// TwinCAT 3 PLC project Panels
// ProgramVersion: 3.1.4026.20
// libraries:
//   Core, * (Beckhoff Automation LLC)
//   CoreComponents, * (Beckhoff Automation LLC)
//   CoreMotionNc2, * (Beckhoff Automation LLC)
//   Mechatronics Core, * (Beckhoff Automation LLC)
//   Tc2_Standard, * (Beckhoff Automation GmbH)
//   Tc2_System, * (Beckhoff Automation GmbH)
//   Xts Core, * (Beckhoff Automation LLC)
// project tree:
//   DUTs/ ST_Chiller_HMI.TcDUT, ST_Compressor_HMI.TcDUT, ST_Conveyor_HMI.TcDUT, ST_CuringOven_HMI.TcDUT, ST_Dispenser_HMI.TcDUT, ST_EStop_HMI.TcDUT, ST_HeaterCooler_HMI.TcDUT, ST_IndexingTable_HMI.TcDUT, ST_InterlockChain_HMI.TcDUT, ST_LightCurtain_HMI.TcDUT, ST_MixingStation_HMI.TcDUT, ST_NetworkSwitch_HMI.TcDUT, ST_LocalLog.TcDUT, ST_PidController_HMI.TcDUT, ST_PeekerEntry.TcDUT, ST_PickAndPlaceUnit_HMI.TcDUT, ST_Pump_HMI.TcDUT, ST_Robot_HMI.TcDUT, ST_SafetyDoor_HMI.TcDUT, ST_UPS_HMI.TcDUT, ST_Valve_HMI.TcDUT, ST_VFD_HMI.TcDUT, ST_Vision_HMI.TcDUT, ST_XtsSystem_HMI.TcDUT, ST_XtsMover_HMI.TcDUT, ST_XtsStation_HMI.TcDUT, ST_XtsPositionTrigger_HMI.TcDUT, ST_XtsZone_HMI.TcDUT
//   / PlcTask.TcTTO
//   POUs/ MAIN.TcPOU
// real-time tasks:
//   TASK PlcTask: cycle T#10ms, priority 20, ADS port 350

CONFIGURATION Panels
    RESOURCE PLC ON TwinCAT3
        TASK PlcTask(INTERVAL := T#10ms, PRIORITY := 20);
        PROGRAM MAIN WITH PlcTask : MAIN;
    END_RESOURCE
END_CONFIGURATION

// ---- DUTs/ST_Chiller_HMI.TcDUT
TYPE ST_Chiller_HMI EXTENDS ST_HmiFunction :
STRUCT

    // Display Parameters - Panel Data Points
    Temperature         : LREAL;        // Current outlet temperature in °C
    FlowRate            : LREAL;        // Current flow rate in L/min

    // Display Parameters - Popup Data Points
    TemperatureSetpoint : LREAL;        // Temperature setpoint in °C
    AlarmStatus         : BOOL;         // Alarm condition present
    InletTemperature    : LREAL;        // Inlet temperature in °C

    // Status Indicators
    Running             : BOOL;         // Chiller is running
    Enabled             : BOOL;         // Chiller is enabled
    HasFault            : BOOL;         // Fault condition present
    AtSetpoint          : BOOL;         // Target setpoint reached
    LowFlowAlarm        : BOOL;         // Low flow alarm active

    // Fault Information
    ErrorId             : DINT;         // Active error code

    // Control Setpoints
    TargetTemperature   : LREAL;        // Target temperature setpoint in °C
    TargetFlowRate      : LREAL;        // Target flow rate in L/min
    MinTemperature      : LREAL;        // Minimum temperature limit in °C
    MaxTemperature      : LREAL;        // Maximum temperature limit in °C

    // Command Buttons (rising edge triggered)
    Start               : Button;       // Start chiller command
    Stop                : Button;       // Stop chiller command
    Reset               : Button;       // Reset fault command

    // Statistics
    TotalRuntime        : LREAL;        // Total runtime in hours
    TotalStarts         : UDINT;        // Total number of starts
    AvgTemperature      : LREAL;        // Average temperature in °C
    AvgFlowRate         : LREAL;        // Average flow rate in L/min
    TotalCoolingEnergy  : LREAL;        // Total cooling energy in kWh
    AlarmCount          : UDINT;        // Total number of alarms

END_STRUCT
END_TYPE

// ---- DUTs/ST_Compressor_HMI.TcDUT
TYPE ST_Compressor_HMI EXTENDS ST_HmiFunction :
STRUCT

    // Display Parameters - Panel Data Points
    Pressure            : LREAL;        // Current pressure in bar
    Runtime             : LREAL;        // Current runtime in hours

    // Display Parameters - Popup Data Points
    MaintenanceInterval : LREAL;        // Next maintenance in hours
    Temperature         : LREAL;        // Current temperature in °C

    // Status Indicators
    Running             : BOOL;         // Compressor is running
    Enabled             : BOOL;         // Compressor is enabled
    HasFault            : BOOL;         // Fault condition present
    AtPressure          : BOOL;         // Target pressure reached
    OverTemperature     : BOOL;         // Temperature limit exceeded

    // Fault Information
    ErrorId             : DINT;         // Active error code

    // Control Setpoints
    TargetPressure      : LREAL;        // Target pressure setpoint in bar
    MaxPressure         : LREAL;        // Maximum pressure limit in bar
    MinPressure         : LREAL;        // Minimum pressure limit in bar
    MaxTemperature      : LREAL;        // Maximum temperature limit in °C

    // Command Buttons (rising edge triggered)
    Start               : Button;       // Start compressor command
    Stop                : Button;       // Stop compressor command
    Reset               : Button;       // Reset fault command

    // Statistics
    TotalStarts         : UDINT;        // Total number of starts
    TotalRuntime        : LREAL;        // Total runtime in hours
    AvgPressure         : LREAL;        // Average pressure in bar
    AvgTemperature      : LREAL;        // Average temperature in °C
    LastMaintenanceDate : STRING;       // Last maintenance date/time
    HoursToMaintenance  : LREAL;        // Hours remaining until maintenance

END_STRUCT
END_TYPE

// ---- DUTs/ST_Conveyor_HMI.TcDUT
TYPE ST_Conveyor_HMI EXTENDS ST_HmiFunction :
STRUCT

	// Status Information
    Running                 : BOOL;           // Conveyor is currently running
    Enabled                 : BOOL;           // Conveyor is enabled
    AutoMode                : BOOL;           // Operating in automatic mode
    JamDetected             : BOOL;           // Jam condition detected
    ReverseDirection        : BOOL;           // Currently running in reverse direction

    // Error Information
    HasError                : BOOL;           // Error condition present
    ErrorCode               : UDINT;          // Specific error code

    // Speed and Motor Information
    ActualSpeed             : LREAL;          // Current conveyor speed
    TargetSpeed             : LREAL;          // Target speed setpoint
    SpeedUnit               : STRING(10);     // Speed unit (e.g., "m/min", "ft/min")
    MotorLoad               : LREAL;          // Motor load percentage (0-100)
    MotorCurrent            : LREAL;          // Motor current in Amps
    MotorTemperature        : LREAL;          // Motor temperature in Celsius

    // Direction Information
    DirectionText           : STRING(20);     // Direction text for display (e.g., "Forward", "Reverse", "Stopped")

    // Tracking and Statistics
    ItemCount               : UDINT;          // Total items transported
    RuntimeHours            : LREAL;          // Total runtime hours
    JamCount                : UDINT;          // Total number of jams detected
    LastJamTime             : STRING(80);     // Timestamp of last jam event

    // Maintenance Information
    MaintenanceDue          : LREAL;          // Hours until maintenance is due
    LastMaintenanceDate     : STRING(80);     // Date of last maintenance
    MaintenanceRequired     : BOOL;           // Maintenance is required
    ResetMaintenance        : BOOL;           // Command to reset maintenance counter

    // Commands (Button type for rising edge detection)
    Start                   : Button;         // Start conveyor command
    Stop                    : Button;         // Stop conveyor command
    Reset                   : Button;         // Reset faults/errors command
    Acknowledge             : Button;         // Acknowledge alarms/warnings command

END_STRUCT
END_TYPE

// ---- DUTs/ST_CuringOven_HMI.TcDUT
{attribute 'qualified_only'}
{attribute 'strict'}
TYPE ST_CuringOven_HMI EXTENDS ST_HmiFunction :
STRUCT
	// Display values
	Zone1Temperature		: LREAL;		// Zone 1 current temperature in °C
	Zone2Temperature		: LREAL;		// Zone 2 current temperature in °C
	Zone3Temperature		: LREAL;		// Zone 3 current temperature in °C
	ConveyorSpeed			: LREAL;		// Current conveyor speed in m/min
	DoorOpen				: BOOL;			// Door open status
	ZonesAtTemperature		: BOOL;			// All zones at target temperature
	Heating					: BOOL;			// Heating active status
	Ready					: BOOL;			// Ready for operation status
    Enabled             : BOOL;         // Dispenser is enabled
    HasFault            : BOOL;         // Fault condition present

    // Fault Information
    ErrorId             : DINT;         // Active error code

	// Control setpoints
	Zone1Setpoint			: LREAL;		// Zone 1 target temperature in °C
	Zone2Setpoint			: LREAL;		// Zone 2 target temperature in °C
	Zone3Setpoint			: LREAL;		// Zone 3 target temperature in °C
	ConveyorSpeedSetpoint	: LREAL;		// Target conveyor speed in m/min
	CureTime				: LREAL;		// Cure time in seconds

	// Command buttons
	Enable					: Button;		// Enable curing oven command
	Disable					: Button;		// Disable curing oven command
	Reset					: Button;		// Reset curing oven command
	OpenDoor				: Button;		// Open door command

	// Statistics
	TotalCycles				: ULINT;		// Total number of curing cycles
	Runtime					: LREAL;		// Total runtime in hours
	AvgCureTime				: LREAL;		// Average cure time in seconds
	EnergyUsed				: LREAL;		// Total energy used in kWh
	LastCycleTime			: LREAL;		// Last cycle time in seconds
END_STRUCT
END_TYPE

// ---- DUTs/ST_Dispenser_HMI.TcDUT
TYPE ST_Dispenser_HMI EXTENDS ST_HmiFunction :
STRUCT

    // Display Parameters - Panel Data Points
    VolumeDispensed     : LREAL;        // Current volume dispensed in mL
    Pressure            : LREAL;        // Current pressure in bar
    NozzleOpen          : BOOL;         // Nozzle open status

    // Display Parameters - Popup Data Points
    FlowRate            : LREAL;        // Current flow rate in mL/s
    Temperature         : LREAL;        // Current temperature in °C

    // Status Indicators
    Enabled             : BOOL;         // Dispenser is enabled
    Dispensing          : BOOL;         // Dispensing in progress
    Ready               : BOOL;         // Ready to dispense
    HasFault            : BOOL;         // Fault condition present

    // Fault Information
    ErrorId             : DINT;         // Active error code

    // Control Setpoints
    TargetVolume        : LREAL;        // Target volume to dispense in mL
    TargetPressure      : LREAL;        // Target pressure in bar
    DispenseTime        : LREAL;        // Target dispense time in seconds
    NozzleSize          : LREAL;        // Nozzle diameter in mm

    // Command Buttons (rising edge triggered)
    Enable              : Button;       // Enable dispenser command
    Disable             : Button;       // Disable dispenser command
    Reset               : Button;       // Reset fault command
    Dispense            : Button;       // Start dispense cycle command

    // Statistics
    TotalDispenses      : UDINT;        // Total number of dispense cycles completed
    TotalVolume         : LREAL;        // Total volume dispensed in liters
    Runtime             : LREAL;        // Total runtime in hours
    AvgDispenseTime     : LREAL;        // Average dispense time in seconds
    LastDispenseVolume  : LREAL;        // Last dispense volume in mL

END_STRUCT
END_TYPE

// ---- DUTs/ST_EStop_HMI.TcDUT
TYPE ST_EStop_HMI EXTENDS ST_HmiFunction :
STRUCT
	
	// Primary Status Indicators
    CircuitOk           : BOOL;           // Emergency stop circuit is intact
    Activated           : BOOL;           // At least one E-Stop button is pressed
    ResetRequired       : BOOL;           // System requires reset after E-Stop activation
    MonitoringActive    : BOOL;           // Safety monitoring is active
    Bypassed            : BOOL;           // Emergency stop circuit is bypassed (dangerous condition)
    
    // Safety System Status
    SafetyRelayOk       : BOOL;           // Safety relay contacts are functioning properly
    RedundancyOk        : BOOL;           // Redundant safety channels are OK
    TestMode            : BOOL;           // System is in test/maintenance mode
    
    // Error Information
    HasError            : BOOL;           // Error condition present
    ErrorCode           : UDINT;          // Specific error code
    
    // Operating Statistics
    ActivationCount     : UDINT;          // Total number of E-Stop activations
    LastActivationTime  : STRING(80);     // Timestamp of last activation
    ResponseTime        : LREAL;          // Last measured response time in milliseconds
    TestCount           : UDINT;          // Number of function tests performed
    LastTestDate        : STRING(80);     // Date/time of last function test
    
    // Bypass Configuration
    BypassTimeout       : UDINT;          // Bypass timeout in seconds (safety feature)
    
    // Distributed E-Stop Stations
    Station1Ok          : BOOL;           // Station 1 E-Stop is not activated and functioning
    Station2Ok          : BOOL;           // Station 2 E-Stop is not activated and functioning
    Station3Ok          : BOOL;           // Station 3 E-Stop is not activated and functioning
    Station4Ok          : BOOL;           // Station 4 E-Stop is not activated and functioning
    TotalStations       : UDINT;          // Total number of E-Stop stations in the system
    ActivatedStationId  : UDINT;          // ID of the station that triggered the E-Stop (0 = none)
    AllStationsOk       : BOOL;           // All configured stations are functioning properly
    
    // Commands (Button type for rising edge detection)
    Reset               : Button;         // Reset the E-Stop system after clearing condition
    Test                : Button;         // Perform a function test of the E-Stop system
    Acknowledge         : Button;         // Acknowledge warning or alarm condition
    
END_STRUCT
END_TYPE

// ---- DUTs/ST_HeaterCooler_HMI.TcDUT
TYPE ST_HeaterCooler_HMI EXTENDS ST_HmiFunction :
STRUCT
	
	// Status Data
    ActualTemperature       : LREAL;          // Current temperature in °C
    TargetTemperature       : LREAL;          // Target/setpoint temperature in °C
    PowerOutput             : LREAL;          // Current power output in %
    EnergyConsumption       : LREAL;          // Total energy consumed in kWh
    
    // Operating Mode
    HeatingMode             : BOOL;           // TRUE = Heating, FALSE = Cooling
    Enabled                 : BOOL;           // System enabled status
    AutoMode                : BOOL;           // TRUE = Auto, FALSE = Manual
    AtSetpoint              : BOOL;           // Temperature at setpoint within tolerance
    
    // Safety & Protection
    ThermalProtectionActive : BOOL;           // Thermal protection triggered
    OverheatAlarm           : BOOL;           // Overheat alarm active
    HasError                : BOOL;           // Error present
    ErrorCode               : UDINT;          // Error code
    
    // Control Parameters
    MaxPowerOutput          : LREAL;          // Maximum power output limit in %
    RampRate                : LREAL;          // Temperature ramp rate in °C/min
    
    // Limits
    TemperatureMax          : LREAL;          // Maximum allowed temperature in °C
    TemperatureMin          : LREAL;          // Minimum allowed temperature in °C
    OverheatTemperature     : LREAL;          // Overheat protection temperature in °C
    TemperatureTolerance    : LREAL;          // Temperature tolerance for at-setpoint in °C
    
    // Commands (buttons)
    Enable                  : Button;
    Disable                 : Button;
    Reset                   : Button;
    Stop                    : Button;
    SwitchMode              : Button;  // Switch between heating and cooling

END_STRUCT
END_TYPE

// ---- DUTs/ST_IndexingTable_HMI.TcDUT
TYPE ST_IndexingTable_HMI EXTENDS ST_HmiFunction :
STRUCT

    // Status and Control
    Enabled                 : BOOL;
    Busy                    : BOOL;
    HasError                : BOOL;
    ErrorCode               : DINT;

    // Position Status
    CurrentPosition         : DINT;             // Current position number (1-based)
    TargetPosition          : DINT;             // Target position number (1-based)
    CurrentPositionName     : STRING(40);       // Name of current position
    TargetPositionName      : STRING(40);       // Name of target position
    PositionCount           : DINT;             // Total number of positions available
    AtPosition              : BOOL;             // True when at target position
    CurrentAngle            : LREAL;            // Current angle in degrees

    // Manual Control Setpoints
    TargetAngle             : LREAL;            // Target angle setpoint in degrees
    RotationSpeedSetpoint   : LREAL;            // Rotation speed setpoint in degrees/second
    ClampPressure           : LREAL;            // Clamp pressure setpoint in bar

    // Rotation
    RotationSpeed           : LREAL;            // Current rotation speed in degrees/second

    // Clamping System
    Clamped                 : BOOL;             // Clamping is active

    // Cycle Data
    IndexCount              : UDINT;            // Total index count
    LastIndexTime           : LREAL;            // Last index time in seconds
    RuntimeHours            : LREAL;            // Total runtime hours

    // Operating Mode
    AutoMode                : BOOL;             // Automatic mode active

    // Commands
    Index                   : Button;           // Index to next position command
    Clamp                   : Button;           // Clamp command
    Unclamp                 : Button;           // Unclamp command
    Home                    : Button;           // Home command
    Reset                   : Button;           // Reset error command

END_STRUCT
END_TYPE

// ---- DUTs/ST_InterlockChain_HMI.TcDUT
TYPE ST_InterlockChain_HMI EXTENDS ST_HmiFunction :
STRUCT

	// Overall Safety Status
    SafetyOk                : BOOL;           // Overall safety chain is satisfied (all conditions met or bypassed)
    AllConditionsMet        : BOOL;           // All active conditions are satisfied without bypass
    MonitoringActive        : BOOL;           // Interlock chain monitoring is active
    Bypassed                : BOOL;           // One or more conditions are bypassed
    LockedOut               : BOOL;           // Chain is locked out and cannot be satisfied

    // Error Information
    HasError                : BOOL;           // Error condition present in the chain
    ErrorCode               : UDINT;          // Specific error code

    // Configuration
    ActiveConditionCount    : UDINT;          // Number of conditions actively monitored (1-6)
    BypassTimeout           : UDINT;          // Bypass timeout in seconds (safety feature)

    // Individual Condition 1
    Condition1Name          : STRING(80);     // Description/name of condition 1
    Condition1Met           : BOOL;           // Condition 1 is satisfied
    Condition1Bypassed      : BOOL;           // Condition 1 is bypassed

    // Individual Condition 2
    Condition2Name          : STRING(80);     // Description/name of condition 2
    Condition2Met           : BOOL;           // Condition 2 is satisfied
    Condition2Bypassed      : BOOL;           // Condition 2 is bypassed

    // Individual Condition 3
    Condition3Name          : STRING(80);     // Description/name of condition 3
    Condition3Met           : BOOL;           // Condition 3 is satisfied
    Condition3Bypassed      : BOOL;           // Condition 3 is bypassed

    // Individual Condition 4
    Condition4Name          : STRING(80);     // Description/name of condition 4
    Condition4Met           : BOOL;           // Condition 4 is satisfied
    Condition4Bypassed      : BOOL;           // Condition 4 is bypassed

    // Individual Condition 5
    Condition5Name          : STRING(80);     // Description/name of condition 5
    Condition5Met           : BOOL;           // Condition 5 is satisfied
    Condition5Bypassed      : BOOL;           // Condition 5 is bypassed

    // Individual Condition 6
    Condition6Name          : STRING(80);     // Description/name of condition 6
    Condition6Met           : BOOL;           // Condition 6 is satisfied
    Condition6Bypassed      : BOOL;           // Condition 6 is bypassed

    // Statistics and Diagnostics
    TotalViolations         : UDINT;          // Total number of times chain was violated
    LastViolationTime       : STRING(80);     // Timestamp of last violation
    ViolatedConditionName   : STRING(80);     // Name of the condition that was last violated
    ChainResponseTime       : LREAL;          // Last measured chain response time in milliseconds
    BypassedConditionCount  : UDINT;          // Current number of bypassed conditions
    EvaluationCount         : UDINT;          // Total number of chain evaluations performed

    // Commands (Button type for rising edge detection)
    Reset                   : Button;         // Reset the interlock chain after violation
    Acknowledge             : Button;         // Acknowledge warning or alarm condition

END_STRUCT
END_TYPE

// ---- DUTs/ST_LightCurtain_HMI.TcDUT
TYPE ST_LightCurtain_HMI EXTENDS ST_HmiFunction :
STRUCT

	// Status Data
    BeamStatus              : BOOL;           // TRUE = Clear, FALSE = Blocked
    MutingActive            : BOOL;           // Muting is currently active
    TestMode                : BOOL;           // System in test mode
    SafetyOutputActive      : BOOL;           // Safety output is active
    
    // Diagnostics
    BeamInterruptionCount   : UDINT;          // Total beam interruptions
    ResponseTime            : LREAL;          // Last response time in ms
    SignalStrength          : LREAL;          // Beam signal strength in %
    LastBeamBreakDuration   : LREAL;          // Duration of last break in seconds
    
    // Operating Data
    OperatingHours          : LREAL;          // Total operating hours
    PowerCycleCount         : UDINT;          // Number of power cycles
    TestCount               : UDINT;          // Number of tests performed
    LastTestDate            : STRING(80);     // Date/time of last test
    
    // Safety & Protection
    HasError                : BOOL;           // Error present
    ErrorCode               : UDINT;          // Error code
    AlarmActive             : BOOL;           // Alarm condition active
    SafetyCircuitOk         : BOOL;           // Safety circuit integrity OK
    ExternalDeviceOk        : BOOL;           // External device monitoring OK
    
    // Muting Configuration
    MutingEnabled           : BOOL;           // Muting function enabled
    MutingTimeout           : UDINT;          // Muting timeout in seconds
    MutingSensorStatus      : BOOL;           // Muting sensors status OK
    
    // System Configuration
    ResolutionCapability    : LREAL;          // Detection capability in mm
    ProtectedHeight         : LREAL;          // Protected field height in mm
    SafetyDistance          : LREAL;          // Minimum safety distance in mm
    
    // Blanking Configuration
    BlankingActive          : BOOL;           // Blanking function active
    BlankingSize            : LREAL;          // Blanking size in mm
    
    // Maintenance
    MaintenanceDue          : LREAL;          // Hours until maintenance
    MaintenanceRequired     : BOOL;           // Maintenance required flag
    LastMaintenanceDate     : STRING(80);     // Last maintenance date
    ResetMaintenance        : BOOL;           // Reset maintenance counter
    
    // Commands (buttons)
    Test                    : Button;         // Perform function test
    Reset                   : Button;         // Reset errors and alarms
    Acknowledge             : Button;         // Acknowledge alarm
    EnableMuting            : Button;         // Enable muting function
    DisableMuting           : Button;         // Disable muting function
    Restart                 : Button;         // Restart device	

END_STRUCT
END_TYPE

// ---- DUTs/ST_MixingStation_HMI.TcDUT
TYPE ST_MixingStation_HMI EXTENDS ST_HmiFunction :
STRUCT

    // Display Parameters - Panel Data Points
    RecipeProgress      : LREAL;        // Recipe completion percentage (0-100%)
    MotorSpeed          : LREAL;        // Current motor speed in RPM

    // Display Parameters - Popup Data Points
    IngredientALevel    : LREAL;        // Ingredient A level percentage (0-100%)
    IngredientBLevel    : LREAL;        // Ingredient B level percentage (0-100%)

    // Status Indicators
    Enabled             : BOOL;         // Station is enabled
    Busy                : BOOL;         // Station is busy processing
    Mixing              : BOOL;         // Mixing process active
    RecipeComplete      : BOOL;         // Recipe completed successfully
    HasFault            : BOOL;         // Fault condition present

    // Fault Information
    ErrorId             : DINT;         // Active error code

    // Control Setpoints
    TargetSpeed         : LREAL;        // Target motor speed in RPM
    MixingTime          : LREAL;        // Target mixing time in seconds
    IngredientATarget   : LREAL;        // Target percentage for Ingredient A (0-100%)
    IngredientBTarget   : LREAL;        // Target percentage for Ingredient B (0-100%)

    // Command Buttons (rising edge triggered)
    Enable              : Button;       // Enable station command
    Disable             : Button;       // Disable station command
    Reset               : Button;       // Reset fault command

    // Statistics
    TotalCycles         : UDINT;        // Total number of mixing cycles completed
    Runtime             : LREAL;        // Total runtime in hours
    LastCycleTime       : LREAL;        // Last cycle time in seconds
    AvgCycleTime        : LREAL;        // Average cycle time in seconds

END_STRUCT
END_TYPE

// ---- DUTs/ST_NetworkSwitch_HMI.TcDUT
TYPE ST_NetworkSwitch_HMI EXTENDS ST_HmiFunction :
STRUCT

    // Display Parameters - Panel Data Points
    PortStatus              : STRING(50);   // Port status text (e.g., "All Up", "1 Down", "2 Down")
    DataThroughput          : REAL;         // Current data throughput in Mbps
    ActivePorts             : DINT;         // Number of active ports
    TotalPorts              : DINT := 24;   // Total number of ports on switch

    // Display Parameters - Popup Data Points
    ErrorRate               : REAL;         // Packet error rate in percent

    // Control Parameters
    MaxBandwidth            : REAL := 1000.0; // Maximum bandwidth per port in Mbps
    VlanId                  : DINT := 1;    // VLAN ID for configuration

    // Status Indicators
    Enabled                 : BOOL;         // Switch is enabled
    Busy                    : BOOL;         // Switch is processing high traffic
    LinkUp                  : BOOL;         // Primary uplink is up
    SpanningTreeActive      : BOOL;         // Spanning tree protocol active
    NetworkCongestion       : BOOL;         // Network experiencing congestion
    PortMirroring           : BOOL;         // Port mirroring enabled
    HasFault                : BOOL;         // Fault condition present

    // Fault Information
    ErrorId                 : DINT;         // Active fault code

    // Command Buttons (rising edge triggered)
    Enable                  : Button;       // Enable switch command
    Disable                 : Button;       // Disable switch command
    Reset                   : Button;       // Reset fault command

    // Statistics
    TotalPackets            : DINT;         // Total packets processed
    DroppedPackets          : DINT;         // Total dropped packets
    TotalErrors             : DINT;         // Total error count
    BroadcastPackets        : DINT;         // Total broadcast packets
    Uptime                  : REAL;         // Switch uptime in hours
    Temperature             : REAL;         // Switch temperature in degrees Celsius

END_STRUCT
END_TYPE

// ---- DUTs/ST_LocalLog.TcDUT
TYPE ST_LocalLog :
STRUCT
    Logs                : ARRAY[0..99] OF STRING(255);  // Array of log message strings
END_STRUCT
END_TYPE

// ---- DUTs/ST_PidController_HMI.TcDUT
TYPE ST_PidController_HMI EXTENDS ST_HmiFunction :
STRUCT
	
	Unit                : STRING(20);           // Unit of measurement (e.g., '°C', 'bar', '%')
    
    // Process Values
    Setpoint            : LREAL;                // Desired value
    ActualValue         : LREAL;                // Current measured value
    Output              : LREAL;                // Controller output (0-100%)
    Error               : LREAL;                // Current error (Setpoint - ActualValue)
    
    // Status
    Enabled             : BOOL;                 // Controller is enabled
    HasError            : BOOL;                 // Error condition present
    ErrorCode           : DINT;                 // Specific error code
    AutoMode            : BOOL;                 // TRUE = Auto, FALSE = Manual
    ReverseActing       : BOOL;                 // TRUE = output decreases as PV increases
    WindupReset         : BOOL;                 // Integral windup reset active
    
    // PID Tuning Parameters
    Kp                  : LREAL;                // Proportional gain
    Ki                  : LREAL;                // Integral gain
    Kd                  : LREAL;                // Derivative gain
    SampleTime          : LREAL;                // Sample time in seconds
    Deadband            : LREAL;                // Error deadband (no action within this range)
    
    // Output Limits
    OutputMax           : LREAL := 100.0;       // Maximum output limit (%)
    OutputMin           : LREAL := 0.0;         // Minimum output limit (%)
    ManualOutput        : LREAL;                // Manual mode output value (%)
    
    // Integral Limits (Anti-windup)
    IntegralMax         : LREAL := 100.0;       // Maximum integral term (%)
    IntegralMin         : LREAL := -100.0;      // Minimum integral term (%)
    
    // Commands (FB_Button structures - pulse on press)
    Enable              : Button;            // Enable controller command
    Disable             : Button;            // Disable controller command
    Reset               : Button;            // Reset controller command
    AutoTune            : Button;            // Start auto-tuning command
    Hold                : Button;            // Hold current output command

END_STRUCT
END_TYPE

// ---- DUTs/ST_PeekerEntry.TcDUT
TYPE ST_PeekerEntry :
STRUCT
    Index               : UINT;           // Peeker index/address
    Value               : LREAL;          // Peeker value
END_STRUCT
END_TYPE

// ---- DUTs/ST_PickAndPlaceUnit_HMI.TcDUT
TYPE ST_PickAndPlaceUnit_HMI EXTENDS ST_HmiFunction :
STRUCT

    // Status and Control
    Enabled                 : BOOL;
    Busy                    : BOOL;
    HasError                : BOOL;
    ErrorCode               : DINT;

    // Position Status
    CurrentPositionName     : STRING(40);       // Name of current position (e.g., "Home", "Pick", "Place")
    TargetPositionName      : STRING(40);       // Name of target position
    AtPosition              : BOOL;             // True when at target position

    // Manual Control Setpoints
    TargetPosition          : DINT;             // Target position number (1-based)
    TargetX                 : LREAL;            // Target X coordinate in mm
    TargetY                 : LREAL;            // Target Y coordinate in mm
    TargetZ                 : LREAL;            // Target Z coordinate in mm
    Speed                   : LREAL;            // Movement speed in mm/s
    VacuumPressureSetpoint  : LREAL;            // Vacuum pressure setpoint in mbar

    // Vacuum System
    VacuumActive            : BOOL;             // Vacuum is currently active
    VacuumPressure          : LREAL;            // Current vacuum pressure in mbar
    VacuumSensorOK          : BOOL;             // Vacuum sensor status
    PartDetected            : BOOL;             // Part detected by vacuum sensor

    // Cycle Data
    CycleCount              : UDINT;            // Total cycle count
    PickCycles              : UDINT;            // Number of pick operations
    PlaceCycles             : UDINT;            // Number of place operations
    LastCycleTime           : LREAL;            // Last cycle time in seconds
    RuntimeHours            : LREAL;            // Total runtime hours

    // Commands
    Pick                    : Button;           // Pick command
    Place                   : Button;           // Place command
    Home                    : Button;           // Home command
    Reset                   : Button;           // Reset error command

END_STRUCT
END_TYPE

// ---- DUTs/ST_Pump_HMI.TcDUT
TYPE ST_Pump_HMI EXTENDS ST_HmiFunction :
STRUCT
    
    // Process Values
    FlowRate            : LREAL;
    FlowUnit            : STRING(20) := 'L/min';
    Pressure            : LREAL;
    PressureUnit        : STRING(20) := 'bar';
    MotorCurrent        : LREAL;
    Speed               : LREAL;  // RPM
    
    // Status
    Running             : BOOL;
    Enabled             : BOOL;
    HasError            : BOOL;
    ErrorCode           : DINT;
    AutoMode            : BOOL;
    AlarmActive         : BOOL;
    
    // Control Setpoints
    TargetSpeed         : LREAL;
    TargetFlowRate      : LREAL;
    
    // Commands
    Start               : Button;
    Stop                : Button;
    Reset               : Button;
    
    // Maintenance Data
    RuntimeHours        : LREAL;
    StartCount          : UDINT;
    MaintenanceDue      : LREAL;  // Hours until maintenance
    LastMaintenanceDate : STRING(20);
    MotorTemperature    : LREAL;  // °C
    VibrationLevel      : LREAL;  // mm/s
    MaintenanceRequired : BOOL;
    ResetMaintenance    : BOOL;	

END_STRUCT
END_TYPE

// ---- DUTs/ST_Robot_HMI.TcDUT
TYPE ST_Robot_HMI EXTENDS ST_HmiFunction :
STRUCT

	// Status Information
    ToolAttached            : BOOL;           // Tool is attached to robot
    ProgramStateText        : STRING(20);     // Program state as text (e.g., "Running", "Stopped", "Paused")
    SafetyOk                : BOOL;           // Safety status is OK
    ProgramRunning          : BOOL;           // Program is currently running
    CurrentProgram          : STRING(80);     // Name of currently loaded/running program

    // Error Information
    HasError                : BOOL;           // Error condition present
    ErrorCode               : UDINT;          // Specific error code
    ErrorText               : STRING(255);    // Error description text

    // Control and Operating State
    Enabled                 : BOOL;           // Robot is enabled
    AutoMode                : BOOL;           // Operating in automatic mode
    Homed                   : BOOL;           // All axes are homed
    Moving                  : BOOL;           // Robot is currently moving
    SpeedOverride           : LREAL;          // Speed override percentage (0-100)
    ToolNumber              : UINT;           // Active tool number

    // Joint Positions (degrees)
    Joint1Position          : LREAL;          // Joint 1 position in degrees
    Joint2Position          : LREAL;          // Joint 2 position in degrees
    Joint3Position          : LREAL;          // Joint 3 position in degrees
    Joint4Position          : LREAL;          // Joint 4 position in degrees
    Joint5Position          : LREAL;          // Joint 5 position in degrees
    Joint6Position          : LREAL;          // Joint 6 position in degrees

    // TCP (Tool Center Point) Position - Cartesian coordinates
    TcpX                    : LREAL;          // TCP X position in mm
    TcpY                    : LREAL;          // TCP Y position in mm
    TcpZ                    : LREAL;          // TCP Z position in mm
    TcpA                    : LREAL;          // TCP A rotation in degrees
    TcpB                    : LREAL;          // TCP B rotation in degrees
    TcpC                    : LREAL;          // TCP C rotation in degrees

    // Statistics and Runtime
    CycleCount              : UDINT;          // Total program cycles completed
    RuntimeHours            : LREAL;          // Total runtime in hours
    LastCycleTime           : LREAL;          // Last cycle time in seconds

    // Commands (Button type for rising edge detection)
    Start                   : Button;         // Start program command
    Stop                    : Button;         // Stop program command
    Home                    : Button;         // Home all axes command
    Reset                   : Button;         // Reset faults/errors command
    Acknowledge             : Button;         // Acknowledge alarms/warnings command

END_STRUCT
END_TYPE

// ---- DUTs/ST_SafetyDoor_HMI.TcDUT
TYPE ST_SafetyDoor_HMI EXTENDS ST_HmiFunction :
STRUCT
    
    // Door Status
    DoorClosed              : BOOL;           // Door is in closed position
    Locked                  : BOOL;           // Door lock is engaged
    Bypassed                : BOOL;           // Safety bypass is active
    
    // Safety System Status
    SafetyCircuitIntegrity  : BOOL;           // Safety circuit integrity check OK
    InterlockOk             : BOOL;           // All interlocks satisfied
    MonitoringActive        : BOOL;           // Safety monitoring active
    EmergencyStopActive     : BOOL;           // Emergency stop circuit active
    
    // Access Control
    AccessGranted           : BOOL;           // Access is currently granted
    AccessDenied            : BOOL;           // Access was denied
    KeySwitchOn             : BOOL;           // Physical key switch in ON position
    GuardLockingActive      : BOOL;           // Guard locking mechanism active
    AccessLevel             : UDINT;          // Required access level (0-10)
    LastAccessUser          : STRING(80);     // Last user who accessed
    LastAccessTime          : STRING(80);     // Timestamp of last access
    
    // Error and Alarm Status
    HasError                : BOOL;           // Error condition present
    ErrorCode               : UDINT;          // Error code if HasError is TRUE
    AlarmActive             : BOOL;           // Alarm condition active
    
    // Operating Data
    DoorOpenCount           : UDINT;          // Total number of door openings
    LockEngageTime          : LREAL;          // Time for lock to engage (seconds)
    BypassTimeout           : UDINT;          // Bypass timeout in seconds
    
    // Commands (Button type for rising edge detection)
    Lock                    : Button;         // Command to lock door
    Unlock                  : Button;         // Command to unlock door
    Acknowledge             : Button;         // Acknowledge alarm/warning
    Reset                   : Button;         // Reset error condition
    
END_STRUCT
END_TYPE

// ---- DUTs/ST_UPS_HMI.TcDUT
TYPE ST_UPS_HMI EXTENDS ST_HmiFunction :
STRUCT

    // Display Parameters - Panel Data Points
    BatteryStatus           : STRING(50);   // Battery status text (e.g., "Normal", "Low", "Critical")
    RuntimeRemaining        : REAL;         // Runtime remaining on battery in minutes
    BatteryCharge           : REAL;         // Battery charge level in percent (0-100)

    // Display Parameters - Popup Data Points
    LoadPercentage          : REAL;         // Current load on UPS in percent (0-100)
    InputVoltage            : REAL;         // Input voltage in Volts
    OutputVoltage           : REAL;         // Output voltage in Volts
    BatteryTemperature      : REAL;         // Battery temperature in degrees Celsius

    // Control Parameters
    LowBatteryThreshold     : REAL := 20.0; // Low battery warning threshold in percent
    ShutdownDelay           : DINT := 300;  // Delay before shutdown in seconds

    // Status Indicators
    Enabled                 : BOOL;         // UPS is enabled
    OnBattery               : BOOL;         // UPS is running on battery power
    Charging                : BOOL;         // Battery is charging
    LowBattery              : BOOL;         // Battery charge below threshold
    Overload                : BOOL;         // UPS is overloaded
    ReplaceBattery          : BOOL;         // Battery needs replacement
    HasFault                : BOOL;         // Fault condition present

    // Fault Information
    ErrorId                 : DINT;         // Active fault code

    // Command Buttons (rising edge triggered)
    Enable                  : Button;       // Enable UPS command
    Disable                 : Button;       // Disable UPS command
    Reset                   : Button;       // Reset fault command

    // Statistics
    TotalBatteryCycles      : DINT;         // Total number of battery charge/discharge cycles
    TotalRuntimeOnBattery   : REAL;         // Total runtime on battery power in hours
    LastPowerOutage         : STRING(50);   // Timestamp of last power outage

END_STRUCT
END_TYPE

// ---- DUTs/ST_Valve_HMI.TcDUT
TYPE ST_Valve_HMI EXTENDS ST_HmiFunction :
STRUCT
	
	// Status and Control
    Enabled : BOOL;
    IsMoving : BOOL;
    HasError : BOOL;
    ErrorCode : UDINT;
    
    // Position and Feedback
    PositionFeedback : LREAL;  // Current position in %
    TargetPosition : LREAL;    // Target position in %
    Speed : LREAL;             // Speed in %/s
    
    // Flow and Pressure
    FlowRate : LREAL;              // Current flow rate
    FlowUnit : STRING(20);         // Flow rate unit (e.g., "L/min", "m³/h")
    PressureDifferential : LREAL;  // Pressure difference across valve
    PressureUnit : STRING(20);     // Pressure unit (e.g., "bar", "psi")
    
    // State Indicators
    AutoMode : BOOL;       // Automatic control mode active
    FullyOpen : BOOL;      // Valve is fully open
    FullyClosed : BOOL;    // Valve is fully closed
    
    // Cycle and Operating Data
    CycleCount : UDINT;           // Number of open/close cycles
    OperatingHours : LREAL;       // Total operating hours
    
    // Maintenance
    MaintenanceDue : LREAL;       // Hours until maintenance is due
    MaintenanceRequired : BOOL;   // Maintenance is required
    LastMaintenanceDate : STRING(80);  // Date of last maintenance
    ResetMaintenance : BOOL;      // Command to reset maintenance counter
    
    // Commands
    Open : BOOL;   // Command to open valve
    Close : BOOL;  // Command to close valve
    Stop : BOOL;   // Command to stop valve movement
    Reset : BOOL;  // Command to reset errors
    
END_STRUCT
END_TYPE

// ---- DUTs/ST_VFD_HMI.TcDUT
TYPE ST_VFD_HMI EXTENDS ST_HmiFunction :
STRUCT
	
    // Display Parameters
    Speed               : REAL;         // Actual motor speed in RPM
    Frequency           : REAL;         // Output frequency in Hz
    MotorCurrent        : REAL;         // Motor current in Amperes
    OutputVoltage       : REAL;         // Output voltage in Volts
    
    // Control Parameters
    TargetSpeed         : REAL;         // Target speed setpoint in RPM
    TargetFrequency     : REAL;         // Target frequency setpoint in Hz
    AccelerationTime    : REAL;         // Acceleration ramp time in seconds
    DecelerationTime    : REAL;         // Deceleration ramp time in seconds
    
    // Limit Parameters
    MaxSpeed            : REAL := 3600; // Maximum speed limit in RPM
    MinSpeed            : REAL := 0;    // Minimum speed limit in RPM
    CurrentLimit        : REAL := 10.0; // Current limit in Amperes
    PowerLimit          : REAL := 5.0;  // Power limit in kW
    
    // Status Indicators
    Running             : BOOL;         // Drive is running
    Ready               : BOOL;         // Drive is ready to run
    RemoteMode          : BOOL;         // Drive in remote control mode
    AtSpeed             : BOOL;         // Drive has reached target speed
    OverLimit           : BOOL;         // Current or power limit exceeded
    OverTemperature     : BOOL;         // Drive over temperature
    HasFault            : BOOL;         // Fault condition present
    
    // Fault Information
    ErrorId           : DINT;         // Active fault code
    
    // Command Buttons (rising edge triggered)
    Start               : Button;         // Start command
    Stop                : Button;         // Stop command
    Reset               : Button;         // Reset fault command
	
END_STRUCT
END_TYPE

// ---- DUTs/ST_Vision_HMI.TcDUT
TYPE ST_Vision_HMI EXTENDS ST_HmiFunction :
STRUCT

    // Display Parameters - Panel Data Points
    PassCount           : UDINT;        // Number of passed inspections
    FailCount           : UDINT;        // Number of failed inspections
    Calibrated          : BOOL;         // Camera calibration status

    // Display Parameters - Popup Data Points
    ImageQuality        : REAL;         // Current image quality score (0-100%)

    // Status Indicators
    Enabled             : BOOL;         // Vision system is enabled
    Busy                : BOOL;         // Inspection in progress
    HasFault            : BOOL;         // Fault condition present

    // Fault Information
    ErrorId             : DINT;         // Active error code

    // Control Setpoints
    ExposureTime        : LREAL;        // Camera exposure time in ms
    Gain                : LREAL;        // Camera gain in dB
    Threshold           : LREAL;        // Detection threshold in %
    Brightness          : LREAL;        // Brightness adjustment in %
    Contrast            : LREAL;        // Contrast adjustment in %
    MinQualityThreshold : LREAL;        // Minimum acceptable quality in %

    // Command Buttons (rising edge triggered)
    Enable              : Button;       // Enable vision system command
    Disable             : Button;       // Disable vision system command
    Reset               : Button;       // Reset fault command
    TriggerInspection   : Button;       // Trigger single inspection command
    Calibrate           : Button;       // Start calibration command

    // Statistics
    TotalInspections    : UDINT;        // Total number of inspections completed
    PassRate            : REAL;         // Pass rate in %
    Runtime             : LREAL;        // Total runtime in hours
    AvgInspectionTime   : LREAL;        // Average inspection time in ms
    LastInspectionTime  : LREAL;        // Last inspection time in ms
    AvgQuality          : REAL;         // Average quality score in %
    LastCalibrationDate : STRING;       // Last calibration date/time
    ImagesSaved         : UDINT;        // Number of images saved to disk

END_STRUCT
END_TYPE

// ---- DUTs/ST_XtsSystem_HMI.TcDUT
TYPE ST_XtsSystem_HMI EXTENDS ST_HmiFunction :
STRUCT

	// Status Information
    CurrentTask             : STRING(80);     // Current task being executed
    LastTask                : STRING(80);     // Last completed task
    Enabled                 : BOOL;           // System is enabled
    Busy                    : BOOL;           // System is busy executing a task
    Initialized             : BOOL;           // System has been initialized
    CaGroup                 : UINT;           // Collision Avoidance Group number
    SystemEnabled           : BOOL;           // System enable state
    Simulated               : BOOL;           // System is in simulation mode
	MoversEnabled			: BOOL;

    // Power Supply Status
    Vdc24Okay               : BOOL;           // 24 VDC power supply OK
    Vdc48Okay               : BOOL;           // 48 VDC power supply OK

    // Error Information
    HasError                : BOOL;           // Error condition present
    ErrorId                 : UDINT;          // Specific error ID
    ErrorText               : STRING(255);    // Error description text

    // Peeker Data for diagnostics
    PeekerData              : ARRAY[0..19] OF ST_PeekerEntry;  // Array of peeker values

    // Local Log
    LocalLog                : ST_LocalLog;    // Log messages structure

    // Commands (Button type for rising edge detection)
    Enable                  : Button;         // Enable system command
    Disable                 : Button;         // Disable system command
    Reset                   : Button;         // Reset faults/errors command
    PeekerUp                : Button;         // Increment peeker index
    PeekerDown              : Button;         // Decrement peeker index
    PeekerPageUp            : Button;         // Increment peeker by page
    PeekerPageDown          : Button;         // Decrement peeker by page
    ClearLog                : Button;         // Clear local log command

END_STRUCT
END_TYPE

// ---- DUTs/ST_XtsMover_HMI.TcDUT
TYPE ST_XtsMover_HMI EXTENDS ST_HmiFunction :
STRUCT

	// Status Information
    CurrentTask             : STRING(80);     // Current task being executed
    Position                : LREAL;          // Current mover position in mm
    Velocity                : LREAL;          // Current velocity in mm/s
    Acceleration            : LREAL;          // Current acceleration in mm/s2
    Deceleration            : LREAL;          // Current deceleration in mm/s2
    Jerk                    : LREAL;          // Current jerk in mm/s3

    // State Flags
    Busy                    : BOOL;           // Mover is busy executing a command
    Enabled                 : BOOL;           // Mover is enabled
    Done                    : BOOL;           // Move command completed
    Initialized             : BOOL;           // Mover has been initialized
    AvoidingCollision       : BOOL;           // Mover is avoiding a collision

    // Group Information
    IdentInGroup            : UINT;           // Mover identification number in group
    MoverInGroup            : UINT;           // Mover number in group

    // Commanded Values
    CommandedPosition       : LREAL;          // Commanded position in mm
    CommandedStationName    : STRING(80);     // Name of commanded station

    // Error Information
    HasError                : BOOL;           // Error condition present
    ErrorId                 : UDINT;          // Specific error ID

    // Target Values for Move Commands
    TargetPosition          : LREAL;          // Target position for move commands (mm)
    TargetVelocity          : LREAL;          // Target velocity (mm/s)
    TargetAcceleration      : LREAL;          // Target acceleration (mm/s2)
    TargetDeceleration      : LREAL;          // Target deceleration (mm/s2)
    TargetGap               : LREAL;          // Target gap distance (mm)
    TargetStation           : STRING(80);     // Target station name

    // Local Log
    LocalLog                : ST_LocalLog;    // Log messages structure

    // Jog Commands (Button type for rising edge detection)
    JogBackwardFast         : Button;         // Jog backward fast command
    JogBackwardSlow         : Button;         // Jog backward slow command
    JogForwardSlow          : Button;         // Jog forward slow command
    JogForwardFast          : Button;         // Jog forward fast command

END_STRUCT
END_TYPE

// ---- DUTs/ST_XtsStation_HMI.TcDUT
TYPE ST_XtsStation_HMI EXTENDS ST_HmiFunction :
STRUCT

	// Status Information
    Position                : LREAL;          // Station position in mm
    MoverPresent            : BOOL;           // Mover is present at station
    Enabled                 : BOOL;           // Station is enabled

    // Current Mover Information
    CurrentMoverName        : STRING(80);     // Name of current mover at station
    CurrentMoverId          : UINT;           // ID of current mover at station

    // Station Configuration
    TargetPosition          : LREAL;          // Target position for station (mm)
    NumberMoversEnroute     : UINT;           // Number of movers enroute to station

    // Control Commands (Button type for rising edge detection)
    Enable                  : Button;         // Enable station command
    Disable                 : Button;         // Disable station command

    // Local Log
    LocalLog                : ST_LocalLog;    // Log messages structure

END_STRUCT
END_TYPE

// ---- DUTs/ST_XtsPositionTrigger_HMI.TcDUT
TYPE ST_XtsPositionTrigger_HMI EXTENDS ST_HmiFunction :
STRUCT

	// Status Information
    Position                : LREAL;          // Position trigger location in mm
    MoverPresent            : BOOL;           // Mover is present at trigger position
    Enabled                 : BOOL;           // Position trigger is enabled

    // Current Mover Information
    CurrentMoverName        : STRING(80);     // Name of current mover at trigger
    CurrentMoverId          : UINT;           // ID of current mover at trigger

    // Trigger Configuration
    NumberMoversEnroute  : UINT;           // Number of movers registered to this trigger
    NumberEventsInQueue     : UINT;           // Number of events pending in queue

    // Control Commands
    Enable                  : BOOL;           // Enable position trigger command
    Disable                 : BOOL;           // Disable position trigger command
	TargetPosition: LREAL;

    // Local Log
    LocalLog                : ST_LocalLog;    // Log messages structure

END_STRUCT
END_TYPE

// ---- DUTs/ST_XtsZone_HMI.TcDUT
TYPE ST_XtsZone_HMI EXTENDS ST_HmiFunction :
STRUCT

	// Current Zone Information
    StartPosition           : LREAL;          // Current start position of zone in mm
    EndPosition             : LREAL;          // Current end position of zone in mm
    Length                  : LREAL;          // Length of zone in mm
    NumberMoversInZone      : UINT;           // Number of movers currently in the zone

    // Target Zone Configuration (Editable)
    TargetStartPosition     : LREAL;          // Target start position for zone (mm)
    TargetEndPosition       : LREAL;          // Target end position for zone (mm)

    // Sorted Mover Functionality
    GetSortedMover          : BOOL;           // Command to get sorted mover
    SortedPosition          : ULINT;          // Position index for sorted mover (input)
    SortedMover             : STRING(80);     // Name of sorted mover at specified position

    // Local Log
    LocalLog                : ST_LocalLog;    // Log messages structure

END_STRUCT
END_TYPE

// ---- POUs/MAIN.TcPOU
PROGRAM MAIN
VAR
	Chiller1: ST_Chiller_HMI;
	Compressor1: ST_Compressor_HMI;
	Heater : ST_HeaterCooler_HMI;
	PID: ST_PidController_HMI;
	Pump: ST_Pump_HMI;
	Valve: ST_Valve_HMI;
	VFD: ST_VFD_HMI;
	Vision1: ST_Vision_HMI;
	SafetyDoor: ST_SafetyDoor_HMI;
	LightCurtain: ST_LightCurtain_HMI;
	MixingStation1: ST_MixingStation_HMI;
	EStop: ST_EStop_HMI;
	InterlockChain: ST_InterlockChain_HMI;
	Conveyor: ST_Conveyor_HMI;
	CuringOven1: ST_CuringOven_HMI;
	Dispenser1: ST_Dispenser_HMI;
	Robot: ST_Robot_HMI;
	PickAndPlaceUnit: ST_PickAndPlaceUnit_HMI;
	IndexingTable: ST_IndexingTable_HMI;
	NetworkSwitch1: ST_NetworkSwitch_HMI;
	UPS: ST_UPS_HMI;
	XtsSystem: ST_XtsSystem_HMI;
	XtsMover: ST_XtsMover_HMI;
	XtsStation: ST_XtsStation_HMI;
	XtsPositionTrigger: ST_XtsPositionTrigger_HMI;
	XtsZone: ST_XtsZone_HMI;
END_VAR

END_PROGRAM
